FUNCTION_BLOCK FB_StationMitZuf EXTENDS FB_Station
VAR_INPUT
	ifTeilHolen:			IF_TeilHolen;
END_VAR
VAR_OUTPUT
END_VAR
VAR
	eHolStatus: 			AblaufStatus := AblaufStatus.bereit;
	eStatusGreifer:			StatusGreifer;
	nTeileZaehler:			INT;	
	nAusschussZaehler:		INT;
END_VAR

//********************************************************************************					
//Schrittbetrieb
fbSchrittbetrieb.eHolStatus := eHolStatus;
fbSchrittbetrieb.bAblaufAktiv := fbSchrittbetrieb.bAblaufAktiv OR nTeileZaehler > 0;

//********************************************************************************					
//Handzyklus (Muss Vor SUPER Call sein, damit diese Version vom Hand Zyklus ausgeführt wird)
//IF			bBtnHandZyklus THEN
//	bBtnHandZyklus := FALSE;
//	
//	IF			stStationInfo.bZyklusFertig
//		AND		bRstInPos
//		AND NOT MAIN.bProduzieren THEN
//		IF			MAIN.hatAufnBeiStJob(stStationInfo.nStationsNr) THEN							//Aufnahme will bearbeitet werden (Teile wurden schon bestellt)
//			ifStation.bearbeitenAnfordern(MAIN.getAufnahmeBeiStation(stStationInfo.nStationsNr));	//Aktuelle Aufnahme wird verwendet
//		ELSE																						//Aufnahme will NICHT bearbeitet werden (Teile müssen bestellt werden)
//			MAIN.vorwahlPseudoaufnahme();
//			ifTeilHolen.holenAnfordern();
//			ifStation.bearbeitenAnfordern(Parameter.cAnzAufnahmen+1);								//Pseudoaufnahme wird verwendet
//		END_IF	
//	END_IF
//END_IF

//********************************************************************************					
//Call Basisklasse
SUPER^(stStationInfo := stStationInfo);

//********************************************************************************					
//Ablauf

IF			stStationInfo.bInitBeendet 
	AND NOT stStationInfo.bReset
	AND NOT fbSchrittbetrieb.bInQueue THEN
	
	IF			nTeileZaehler > 0  THEN
		ifTeilHolen.teilHolen();
	END_IF
END_IF


IF			(nAusschussZaehler > 0)
	AND		(nTeileZaehler > 1
	OR		(nTeileZaehler > 0
	AND		(eHolStatus = AblaufStatus.bereit))) THEN
	nTeileZaehler := nTeileZaehler-1;
	nAusschussZaehler := nAusschussZaehler-1;
END_IF

//********************************************************************************
//Statusanzeige
IF			stStationInfo.bInitBeendet
	AND	NOT	stStationInfo.bReset
	AND NOT stStationInfo.bInit
	AND NOT (eStatusGreifer = StatusGreifer.teilGeholt)
	AND NOT (eStatusGreifer = StatusGreifer.teilAbgelegt) THEN	
	stStationInfo.sStatus := TO_STRING(eHolStatus);
END_IF

METHOD ausschussMelden
VAR_INPUT
END_VAR
nAusschussZaehler := nAusschussZaehler+1;
END_METHOD

METHOD holenAnfordern
VAR_INPUT
END_VAR
nTeileZaehler := nTeileZaehler+1;
END_METHOD

END_FUNCTION_BLOCK

(* stored: Version 1.1.0.1, ProductVersion 3.1.4024.12
   POU FB_StationMitZuf: Id {27135f01-859d-4713-8899-53fc55e1cddc}, SpecialFunc None
   Method ausschussMelden: Id {653abd3d-a6e1-4eb4-a649-0a92cf4bf0ff}
   Method holenAnfordern: Id {41960a1e-5c82-47b8-a1c3-262360560cc5} *)
